// SIMATIC S7-200 SMART project (STEP 7-Micro/WIN SMART), CPU SR20

SYMBOL_TABLE 系统符号
Always_On        SM0.0    // 始终接通
Clock_1s         SM0.5    // 针对 1 s 的周期时间，时钟脉冲接通 0.5 s，断开 0.5 s.
END_SYMBOL_TABLE

ORGANIZATION_BLOCK MAIN:OB1
TITLE=程序注释
BEGIN
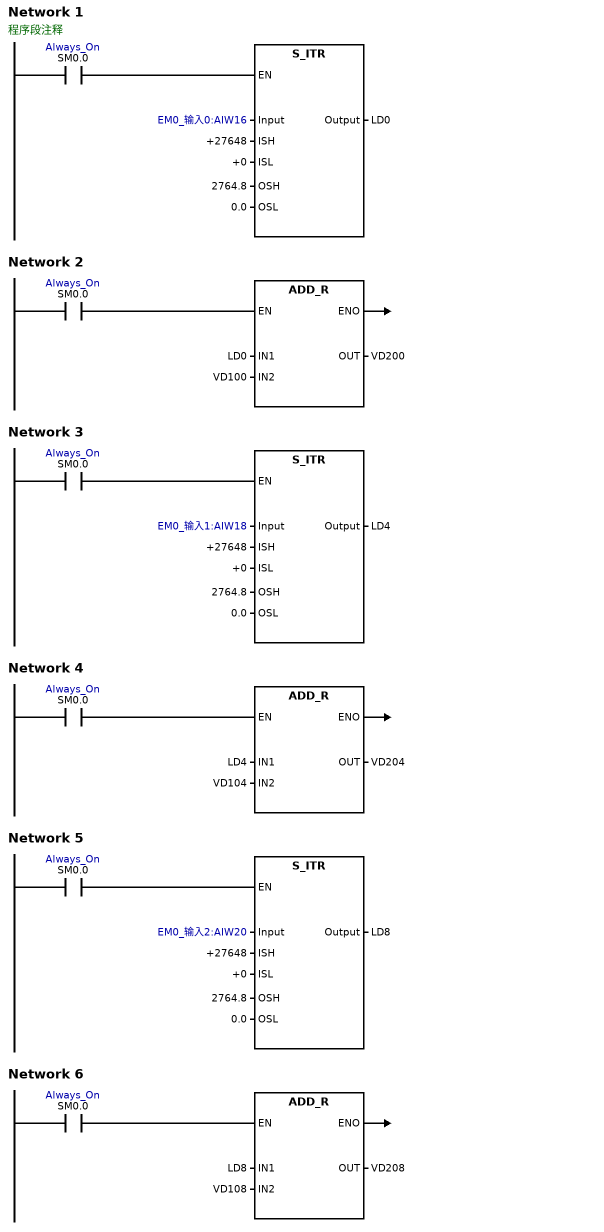
Network 1
// 程序段注释
LD     Always_On:SM0.0
CALL   S_ITR:SBR1, EM0_输入0:AIW16, +27648, +0, 2764.8, 0.0, LD0
Network 2
LD     Always_On:SM0.0
MOVR   LD0, VD200
+R     VD100, VD200
Network 3
LD     Always_On:SM0.0
CALL   S_ITR:SBR1, EM0_输入1:AIW18, +27648, +0, 2764.8, 0.0, LD4
Network 4
LD     Always_On:SM0.0
MOVR   LD4, VD204
+R     VD104, VD204
Network 5
LD     Always_On:SM0.0
CALL   S_ITR:SBR1, EM0_输入2:AIW20, +27648, +0, 2764.8, 0.0, LD8
Network 6
LD     Always_On:SM0.0
MOVR   LD8, VD208
+R     VD108, VD208
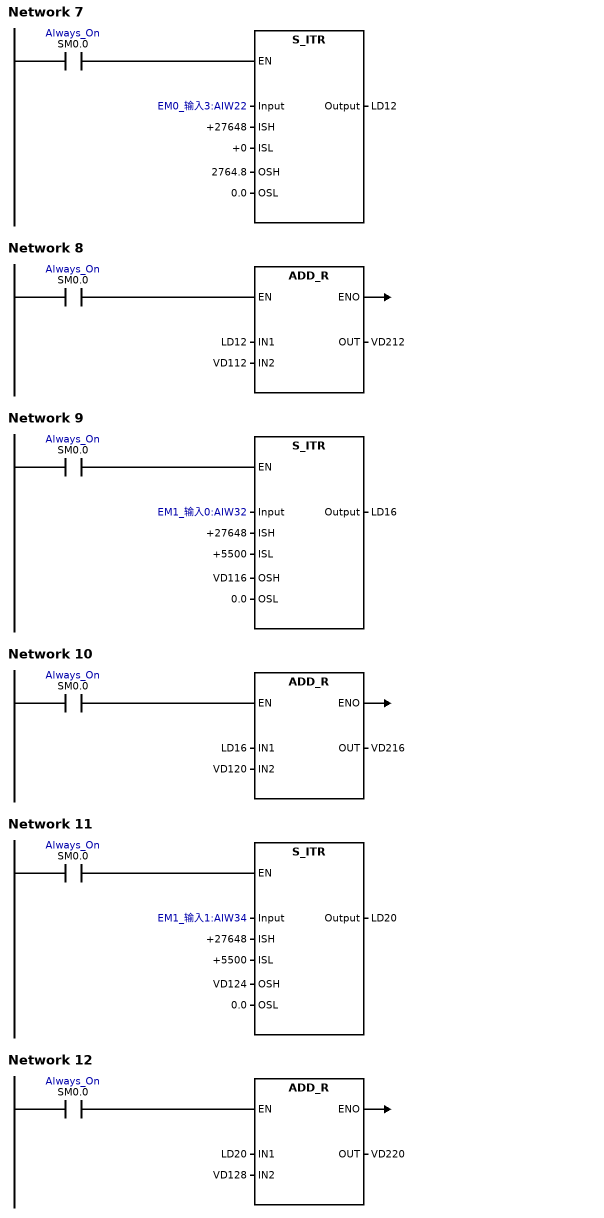
Network 7
LD     Always_On:SM0.0
CALL   S_ITR:SBR1, EM0_输入3:AIW22, +27648, +0, 2764.8, 0.0, LD12
Network 8
LD     Always_On:SM0.0
MOVR   LD12, VD212
+R     VD112, VD212
Network 9
LD     Always_On:SM0.0
CALL   S_ITR:SBR1, EM1_输入0:AIW32, +27648, +5500, VD116, 0.0, LD16
Network 10
LD     Always_On:SM0.0
MOVR   LD16, VD216
+R     VD120, VD216
Network 11
LD     Always_On:SM0.0
CALL   S_ITR:SBR1, EM1_输入1:AIW34, +27648, +5500, VD124, 0.0, LD20
Network 12
LD     Always_On:SM0.0
MOVR   LD20, VD220
+R     VD128, VD220
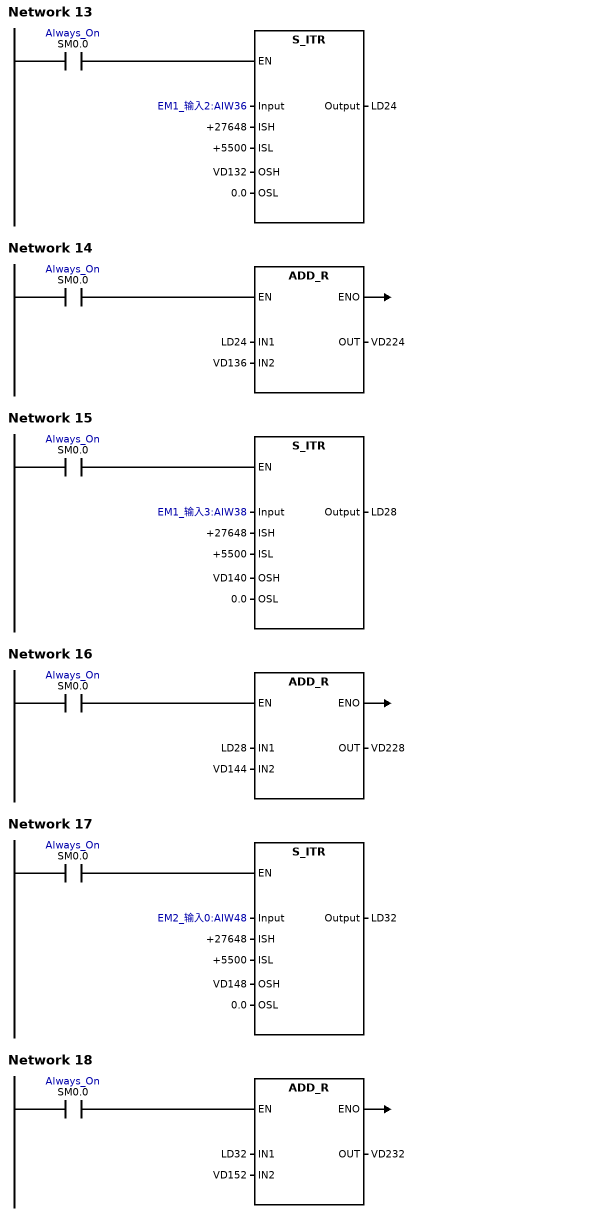
Network 13
LD     Always_On:SM0.0
CALL   S_ITR:SBR1, EM1_输入2:AIW36, +27648, +5500, VD132, 0.0, LD24
Network 14
LD     Always_On:SM0.0
MOVR   LD24, VD224
+R     VD136, VD224
Network 15
LD     Always_On:SM0.0
CALL   S_ITR:SBR1, EM1_输入3:AIW38, +27648, +5500, VD140, 0.0, LD28
Network 16
LD     Always_On:SM0.0
MOVR   LD28, VD228
+R     VD144, VD228
Network 17
LD     Always_On:SM0.0
CALL   S_ITR:SBR1, EM2_输入0:AIW48, +27648, +5500, VD148, 0.0, LD32
Network 18
LD     Always_On:SM0.0
MOVR   LD32, VD232
+R     VD152, VD232
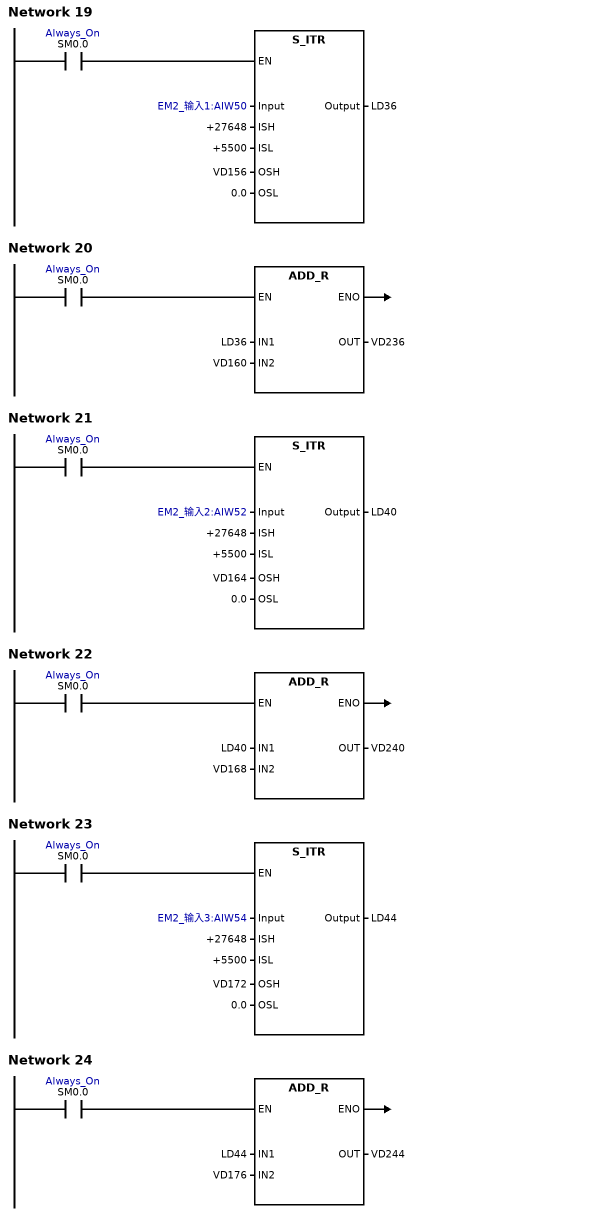
Network 19
LD     Always_On:SM0.0
CALL   S_ITR:SBR1, EM2_输入1:AIW50, +27648, +5500, VD156, 0.0, LD36
Network 20
LD     Always_On:SM0.0
MOVR   LD36, VD236
+R     VD160, VD236
Network 21
LD     Always_On:SM0.0
CALL   S_ITR:SBR1, EM2_输入2:AIW52, +27648, +5500, VD164, 0.0, LD40
Network 22
LD     Always_On:SM0.0
MOVR   LD40, VD240
+R     VD168, VD240
Network 23
LD     Always_On:SM0.0
CALL   S_ITR:SBR1, EM2_输入3:AIW54, +27648, +5500, VD172, 0.0, LD44
Network 24
LD     Always_On:SM0.0
MOVR   LD44, VD244
+R     VD176, VD244
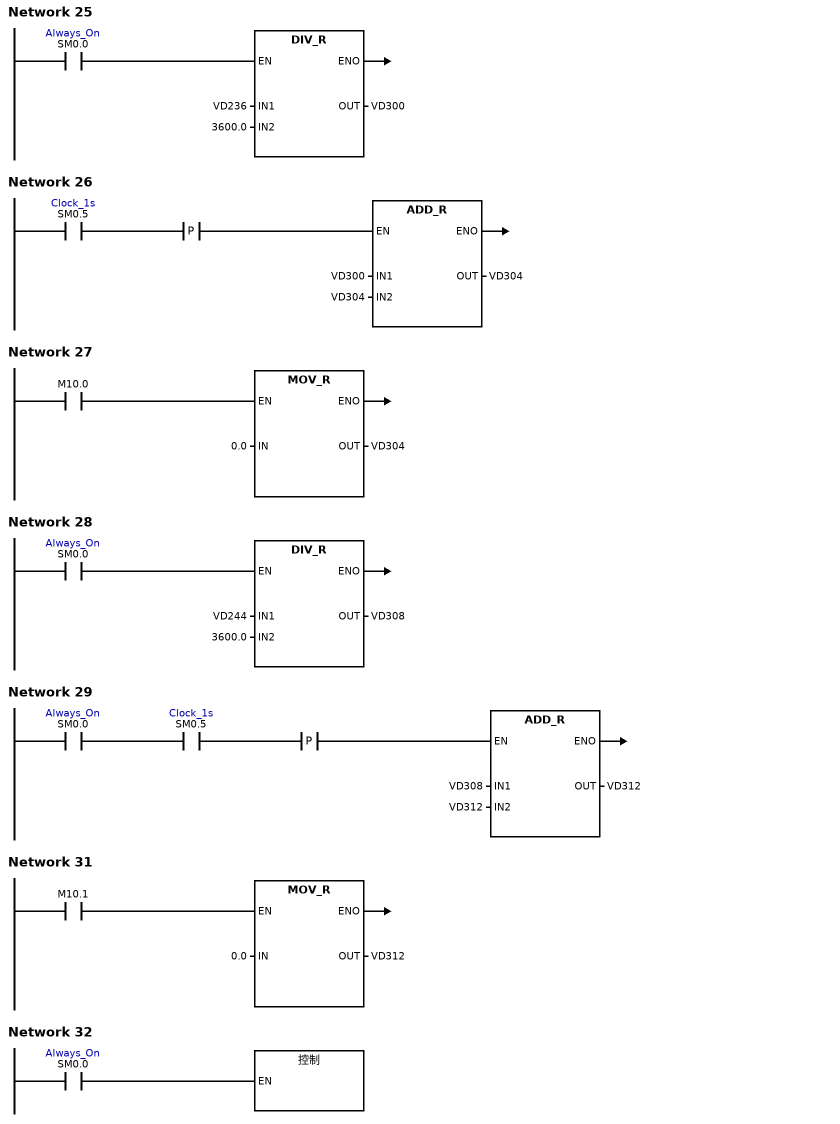
Network 25
LD     Always_On:SM0.0
MOVR   VD236, VD300
/R     3600.0, VD300
Network 26
LD     Clock_1s:SM0.5
EU
+R     VD300, VD304
Network 27
LD     M10.0
MOVR   0.0, VD304
Network 28
LD     Always_On:SM0.0
MOVR   VD244, VD308
/R     3600.0, VD308
Network 29
LD     Always_On:SM0.0
A      Clock_1s:SM0.5
EU
+R     VD308, VD312
Network 31
LD     M10.1
MOVR   0.0, VD312
Network 32
LD     Always_On:SM0.0
CALL   控制:SBR0
END_ORGANIZATION_BLOCK

SUBROUTINE_BLOCK 控制:SBR0
TITLE=子程序注释
BEGIN
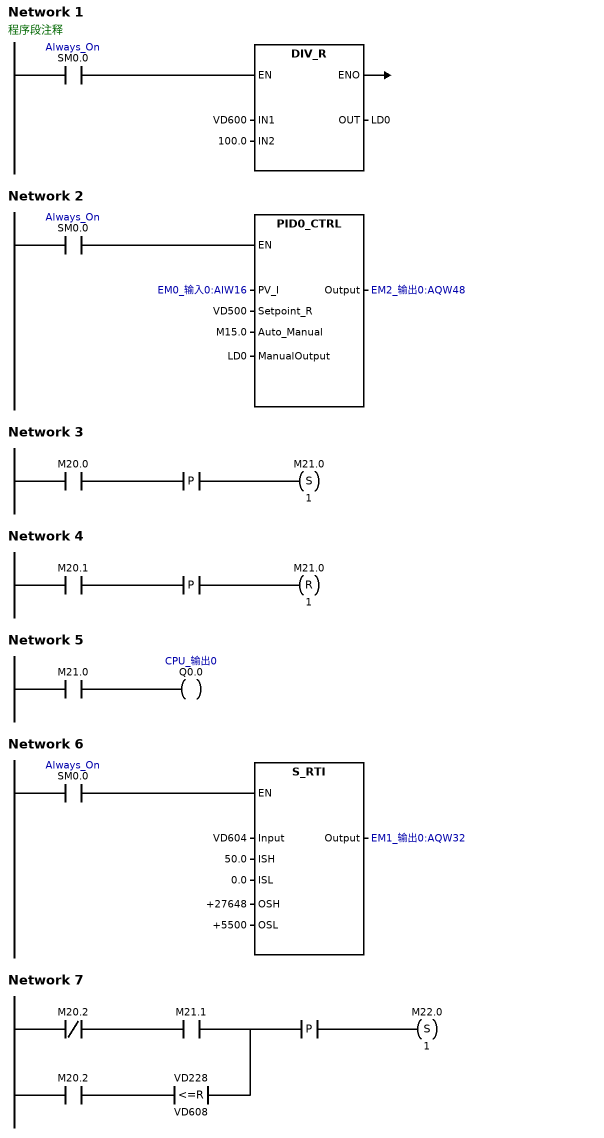
Network 1
// 程序段注释
LD     Always_On:SM0.0
MOVR   VD600, LD0
/R     100.0, LD0
Network 2
LD     Always_On:SM0.0
CALL   PID0_CTRL:SBR2, EM0_输入0:AIW16, VD500, M15.0, LD0, EM2_输出0:AQW48
Network 3
LD     M20.0
EU
S      M21.0, 1
Network 4
LD     M20.1
EU
R      M21.0, 1
Network 5
LD     M21.0
=      CPU_输出0:Q0.0
Network 6
LD     Always_On:SM0.0
CALL   S_RTI:SBR3, VD604, 50.0, 0.0, +27648, +5500, EM1_输出0:AQW32
Network 7
LDN    M20.2
A      M21.1
LD     M20.2
AR<=   VD228, VD608
OLD
EU
S      M22.0, 1
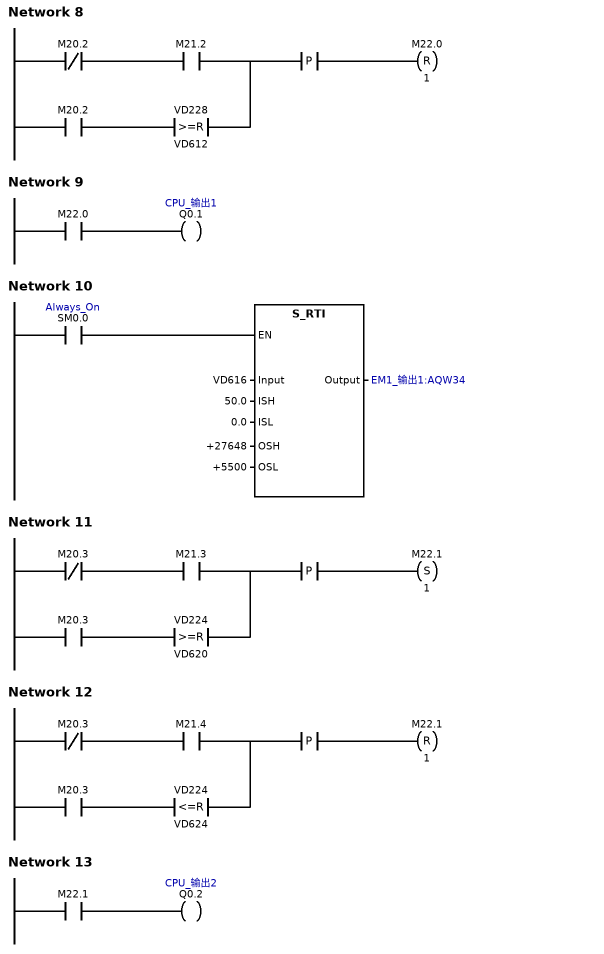
Network 8
LDN    M20.2
A      M21.2
LD     M20.2
AR>=   VD228, VD612
OLD
EU
R      M22.0, 1
Network 9
LD     M22.0
=      CPU_输出1:Q0.1
Network 10
LD     Always_On:SM0.0
CALL   S_RTI:SBR3, VD616, 50.0, 0.0, +27648, +5500, EM1_输出1:AQW34
Network 11
LDN    M20.3
A      M21.3
LD     M20.3
AR>=   VD224, VD620
OLD
EU
S      M22.1, 1
Network 12
LDN    M20.3
A      M21.4
LD     M20.3
AR<=   VD224, VD624
OLD
EU
R      M22.1, 1
Network 13
LD     M22.1
=      CPU_输出2:Q0.2
END_SUBROUTINE_BLOCK

// SBR1: protected block, not included

// SBR2: protected block, not included

// SBR3: protected block, not included

// INT1: protected block, not included
